TYPE ST_Name :
STRUCT
(**轴**)
	AnAxisNo:      ST_AxisName;  //正极
	CaAxisNo:      ST_AxisName;//负极
	
    AnVirAxisNo:      ST_VirAxisName;//正极
	CaVirAxisNo:      ST_VirAxisName;//负极
	VirTimeWind:INT;//模切虚拟摆杆放卷轴 
(**气缸**)
	AnCYNo:        ST_CylinderName;//正极
	CaCYNo:        ST_CylinderName;//负极

(**电磁阀**)
	AnEVNo:        ST_ElectValveName;//正极
	CaEVNo:        ST_ElectValveName;//负极

(***纠偏**)
    AnRecNo:         ST_RecName;//正极
	CaRecNo:         ST_RecName;//负极

(***凸轮表号**)
	 AnTableNo:  ST_TableNo;// 正极
	 CaTableNo:  ST_TableNo;// 负极
	 
(***除尘电机号**)
	 AnMotorNo:  ST_MotorName;// 正极
	 CaMotorNo:  ST_MotorName;// 负极

(***数据工位号**)	 
	 AnBeltNo:ST_BeltNo;//正极
	 CaBeltNo:ST_BeltNo;//负极
	 AnTabNo:ST_TabNo;//正极
	 CaTabNo:ST_TabNo;//负极
	 AnIntervalNo:ST_IntervalNo;//正极
	 CaIntervalNo:ST_IntervalNo;//负极
END_STRUCT
END_TYPE

(* stored: Version 1.1.0.1, ProductVersion 3.1.4024.9
   DUT ST_Name: Id {c6e9295d-c555-44a4-ba2f-bc631cf3746f} *)
